FUNCTION_BLOCK FB_Valve EXTENDS FB_Base IMPLEMENTS I_Valve
VAR_INPUT
END_VAR
VAR_OUTPUT
END_VAR
VAR
END_VAR

METHOD MoveToHome : BOOL
VAR_INPUT
END_VAR
Tc2_System.ADSLOGSTR(0, 'valve move to home', '');

MoveToHome := TRUE;
END_METHOD

METHOD MoveToWork : BOOL
VAR_INPUT
END_VAR
Tc2_System.ADSLOGSTR(0, 'valve move to work', '');

MoveToWork := TRUE;
END_METHOD

END_FUNCTION_BLOCK

(* stored: Version 1.1.0.1
   POU FB_Valve: Id {530fbcc6-073c-4f99-a235-ea2b7e45a87d}, SpecialFunc None
   Method MoveToHome: Id {a3b2d830-9e2d-4c42-9c66-dcf8ffc96541}
   Method MoveToWork: Id {9d596b34-086c-4c11-b355-243d5fd015ff} *)
